TYPE ID_Decoded_DUT :
STRUCT
	Device_Type:  INT;
	Level:  INT;
	VTD:  INT;
END_STRUCT
END_TYPE

(* stored: Version 1.1.0.1
   DUT ID_Decoded_DUT: Id {4e44c35c-cf95-45ba-aca2-dfe7b8d3da93} *)
